KUKA KRL program: Station500_SprueCutter.src, Station500_SprueCutter.dat

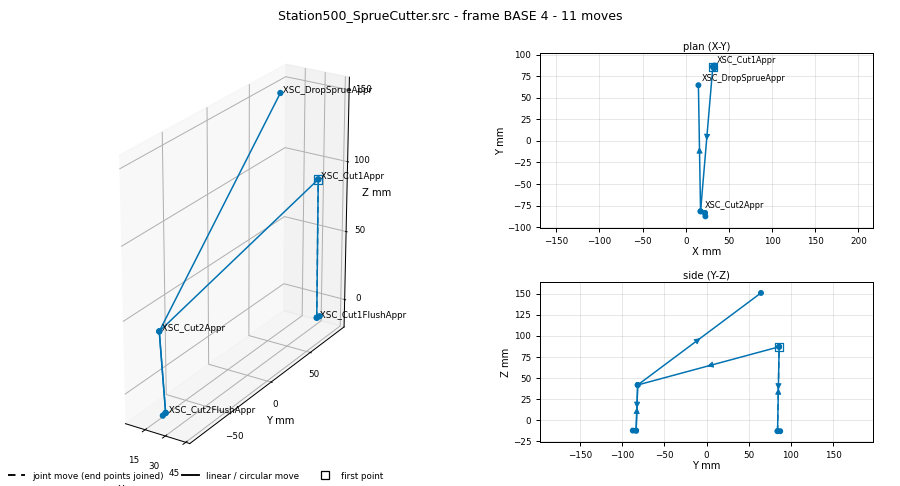
[picture p0: tool path of Station500_SprueCutter.src in frame BASE 4, 11 of 18 moves have a stored position in this frame; points joined in program order, loops and branches not executed]
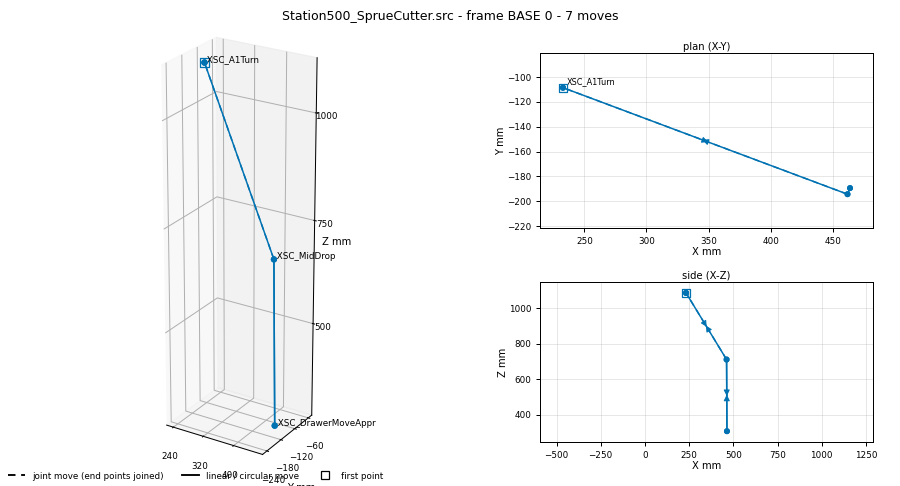
[picture p1: tool path of Station500_SprueCutter.src in frame BASE 0, 7 of 18 moves have a stored position in this frame; points joined in program order, loops and branches not executed]
--- Station500_SprueCutter.src ---
&ACCESS RVO1
&REL 8
&PARAM DISKPATH = KRC:\R1\Program
DEF Station500_SprueCutter()
   ;FOLD INI;%{PE}
      ;FOLD BASISTECH INI
         GLOBAL INTERRUPT DECL 3 WHEN $STOPMESS == TRUE DO IR_STOPM()
         INTERRUPT ON 3
         BAS(#INITMOV, 0)
      ;ENDFOLD (BASISTECH INI)
      ;FOLD USER INI
         ;Make your modifications here
      ;ENDFOLD (USER INI)
   ;ENDFOLD (INI)
;FOLD SPTP SC_A1Turn Vel=100 % PDAT2 Tool[0] Base[0] ;%{PE}
;FOLD Parameters ;%{h}
;Params IlfProvider=kukaroboter.basistech.inlineforms.movement.spline; Kuka.IsGlobalPoint=False; Kuka.PointName=SC_A1Turn; Kuka.BlendingEnabled=False; Kuka.MoveDataPtpName=PDAT2; Kuka.VelocityPtp=100; Kuka.VelocityFieldEnabled=True; Kuka.ColDetectFieldEnabled=True; Kuka.CurrentCDSetIndex=0; Kuka.MovementParameterFieldEnabled=True; IlfCommand=SPTP
;ENDFOLD
SPTP XSC_A1Turn WITH $VEL_AXIS[1] = SVEL_JOINT(100.0), $TOOL = STOOL2(FSC_A1Turn), $BASE = SBASE(FSC_A1Turn.BASE_NO), $IPO_MODE = SIPO_MODE(FSC_A1Turn.IPO_FRAME), $LOAD = SLOAD(FSC_A1Turn.TOOL_NO), $ACC_AXIS[1] = SACC_JOINT(PPDAT2), $APO = SAPO_PTP(PPDAT2), $GEAR_JERK[1] = SGEAR_JERK(PPDAT2), $COLLMON_TOL_PRO[1] = USE_CM_PRO_VALUES(0)
;ENDFOLD

   ;FOLD SPTP SC_Cut1Appr Vel=100 % PDAT4 Tool[2]:TOOL_DATA[2] Base[4]:BASE_DATA[4] ;%{PE}
      ;FOLD Parameters ;%{h}
         ;Params IlfProvider=kukaroboter.basistech.inlineforms.movement.spline; Kuka.IsGlobalPoint=False; Kuka.PointName=SC_Cut1Appr; Kuka.BlendingEnabled=False; Kuka.MoveDataPtpName=PDAT4; Kuka.VelocityPtp=100; Kuka.VelocityFieldEnabled=True; Kuka.ColDetectFieldEnabled=True; Kuka.CurrentCDSetIndex=0; Kuka.MovementParameterFieldEnabled=True; IlfCommand=SPTP; SimId=
      ;ENDFOLD
      SPTP XSC_Cut1Appr WITH $VEL_AXIS[1] = SVEL_JOINT(100.0), $TOOL = STOOL2(FSC_Cut1Appr), $BASE = SBASE(FSC_Cut1Appr.BASE_NO), $IPO_MODE = SIPO_MODE(FSC_Cut1Appr.IPO_FRAME), $LOAD = SLOAD(FSC_Cut1Appr.TOOL_NO), $ACC_AXIS[1] = SACC_JOINT(PPDAT4), $APO = SAPO_PTP(PPDAT4), $GEAR_JERK[1] = SGEAR_JERK(PPDAT4), $COLLMON_TOL_PRO[1] = USE_CM_PRO_VALUES(0)
      ;ENDFOLD

   ;FOLD SLIN SC_Cut1FlushAppr Vel=0.2 m/s CPDAT8 Tool[2]:TOOL_DATA[2] Base[4]:BASE_DATA[4] ;%{PE}
      ;FOLD Parameters ;%{h}
         ;Params IlfProvider=kukaroboter.basistech.inlineforms.movement.spline; Kuka.IsGlobalPoint=False; Kuka.PointName=SC_Cut1FlushAppr; Kuka.BlendingEnabled=False; Kuka.MoveDataName=CPDAT8; Kuka.VelocityPath=0.2; Kuka.VelocityFieldEnabled=True; Kuka.ColDetectFieldEnabled=True; Kuka.CurrentCDSetIndex=0; Kuka.MovementParameterFieldEnabled=True; IlfCommand=SLIN; SimId=
      ;ENDFOLD
      SLIN XSC_Cut1FlushAppr WITH $VEL = SVEL_CP(0.2, , LCPDAT8), $TOOL = STOOL2(FSC_Cut1FlushAppr), $BASE = SBASE(FSC_Cut1FlushAppr.BASE_NO), $IPO_MODE = SIPO_MODE(FSC_Cut1FlushAppr.IPO_FRAME), $LOAD = SLOAD(FSC_Cut1FlushAppr.TOOL_NO), $ACC = SACC_CP(LCPDAT8), $ORI_TYPE = SORI_TYP(LCPDAT8), $APO = SAPO(LCPDAT8), $JERK = SJERK(LCPDAT8), $COLLMON_TOL_PRO[1] = USE_CM_PRO_VALUES(0)
      ;ENDFOLD

   ;FOLD SLIN SC_Cut1Flush Vel=0.1 m/s CPDAT5 Tool[2]:TOOL_DATA[2] Base[4]:BASE_DATA[4] ;%{PE}
      ;FOLD Parameters ;%{h}
         ;Params IlfProvider=kukaroboter.basistech.inlineforms.movement.spline; Kuka.IsGlobalPoint=False; Kuka.PointName=SC_Cut1Flush; Kuka.BlendingEnabled=False; Kuka.MoveDataName=CPDAT5; Kuka.VelocityPath=0.1; Kuka.VelocityFieldEnabled=True; Kuka.ColDetectFieldEnabled=True; Kuka.CurrentCDSetIndex=0; Kuka.MovementParameterFieldEnabled=True; IlfCommand=SLIN; SimId=
      ;ENDFOLD
      SLIN XSC_Cut1Flush WITH $VEL = SVEL_CP(0.1, , LCPDAT5), $TOOL = STOOL2(FSC_Cut1Flush), $BASE = SBASE(FSC_Cut1Flush.BASE_NO), $IPO_MODE = SIPO_MODE(FSC_Cut1Flush.IPO_FRAME), $LOAD = SLOAD(FSC_Cut1Flush.TOOL_NO), $ACC = SACC_CP(LCPDAT5), $ORI_TYPE = SORI_TYP(LCPDAT5), $APO = SAPO(LCPDAT5), $JERK = SJERK(LCPDAT5), $COLLMON_TOL_PRO[1] = USE_CM_PRO_VALUES(0)
      ;ENDFOLD

RtoPLC_SprueCut1=True
    Wait Sec .25
RtoPLC_SprueCut1=False
    Wait Sec .25
   ;FOLD SLIN SC_Cut1FlushAppr Vel=0.2 m/s CPDAT8 Tool[2]:TOOL_DATA[2] Base[4]:BASE_DATA[4] ;%{PE}
      ;FOLD Parameters ;%{h}
         ;Params IlfProvider=kukaroboter.basistech.inlineforms.movement.spline; Kuka.IsGlobalPoint=False; Kuka.PointName=SC_Cut1FlushAppr; Kuka.BlendingEnabled=False; Kuka.MoveDataName=CPDAT8; Kuka.VelocityPath=0.2; Kuka.VelocityFieldEnabled=True; Kuka.ColDetectFieldEnabled=True; Kuka.CurrentCDSetIndex=0; Kuka.MovementParameterFieldEnabled=True; IlfCommand=SLIN; SimId=
      ;ENDFOLD
      SLIN XSC_Cut1FlushAppr WITH $VEL = SVEL_CP(0.2, , LCPDAT8), $TOOL = STOOL2(FSC_Cut1FlushAppr), $BASE = SBASE(FSC_Cut1FlushAppr.BASE_NO), $IPO_MODE = SIPO_MODE(FSC_Cut1FlushAppr.IPO_FRAME), $LOAD = SLOAD(FSC_Cut1FlushAppr.TOOL_NO), $ACC = SACC_CP(LCPDAT8), $ORI_TYPE = SORI_TYP(LCPDAT8), $APO = SAPO(LCPDAT8), $JERK = SJERK(LCPDAT8), $COLLMON_TOL_PRO[1] = USE_CM_PRO_VALUES(0)
      ;ENDFOLD

   ;FOLD SPTP SC_Cut1Appr Vel=100 % PDAT4 Tool[2]:TOOL_DATA[2] Base[4]:BASE_DATA[4] ;%{PE}
      ;FOLD Parameters ;%{h}
         ;Params IlfProvider=kukaroboter.basistech.inlineforms.movement.spline; Kuka.IsGlobalPoint=False; Kuka.PointName=SC_Cut1Appr; Kuka.BlendingEnabled=False; Kuka.MoveDataPtpName=PDAT4; Kuka.VelocityPtp=100; Kuka.VelocityFieldEnabled=True; Kuka.ColDetectFieldEnabled=True; Kuka.CurrentCDSetIndex=0; Kuka.MovementParameterFieldEnabled=True; IlfCommand=SPTP; SimId=
      ;ENDFOLD
      SPTP XSC_Cut1Appr WITH $VEL_AXIS[1] = SVEL_JOINT(100.0), $TOOL = STOOL2(FSC_Cut1Appr), $BASE = SBASE(FSC_Cut1Appr.BASE_NO), $IPO_MODE = SIPO_MODE(FSC_Cut1Appr.IPO_FRAME), $LOAD = SLOAD(FSC_Cut1Appr.TOOL_NO), $ACC_AXIS[1] = SACC_JOINT(PPDAT4), $APO = SAPO_PTP(PPDAT4), $GEAR_JERK[1] = SGEAR_JERK(PPDAT4), $COLLMON_TOL_PRO[1] = USE_CM_PRO_VALUES(0)
      ;ENDFOLD

   ;FOLD SLIN SC_Cut2Appr Vel=2 m/s CPDAT3 Tool[2]:TOOL_DATA[2] Base[4]:BASE_DATA[4] ;%{PE}
      ;FOLD Parameters ;%{h}
         ;Params IlfProvider=kukaroboter.basistech.inlineforms.movement.spline; Kuka.IsGlobalPoint=False; Kuka.PointName=SC_Cut2Appr; Kuka.BlendingEnabled=False; Kuka.MoveDataName=CPDAT3; Kuka.VelocityPath=2; Kuka.VelocityFieldEnabled=True; Kuka.ColDetectFieldEnabled=True; Kuka.CurrentCDSetIndex=0; Kuka.MovementParameterFieldEnabled=True; IlfCommand=SLIN; SimId=
      ;ENDFOLD
      SLIN XSC_Cut2Appr WITH $VEL = SVEL_CP(2.0, , LCPDAT3), $TOOL = STOOL2(FSC_Cut2Appr), $BASE = SBASE(FSC_Cut2Appr.BASE_NO), $IPO_MODE = SIPO_MODE(FSC_Cut2Appr.IPO_FRAME), $LOAD = SLOAD(FSC_Cut2Appr.TOOL_NO), $ACC = SACC_CP(LCPDAT3), $ORI_TYPE = SORI_TYP(LCPDAT3), $APO = SAPO(LCPDAT3), $JERK = SJERK(LCPDAT3), $COLLMON_TOL_PRO[1] = USE_CM_PRO_VALUES(0)
      ;ENDFOLD

   ;FOLD SLIN SC_Cut2FlushAppr Vel=0.2 m/s CPDAT10 Tool[2]:TOOL_DATA[2] Base[4]:BASE_DATA[4] ;%{PE}
      ;FOLD Parameters ;%{h}
         ;Params IlfProvider=kukaroboter.basistech.inlineforms.movement.spline; Kuka.IsGlobalPoint=False; Kuka.PointName=SC_Cut2FlushAppr; Kuka.BlendingEnabled=False; Kuka.MoveDataName=CPDAT10; Kuka.VelocityPath=0.2; Kuka.VelocityFieldEnabled=True; Kuka.ColDetectFieldEnabled=True; Kuka.CurrentCDSetIndex=0; Kuka.MovementParameterFieldEnabled=True; IlfCommand=SLIN; SimId=
      ;ENDFOLD
      SLIN XSC_Cut2FlushAppr WITH $VEL = SVEL_CP(0.2, , LCPDAT10), $TOOL = STOOL2(FSC_Cut2FlushAppr), $BASE = SBASE(FSC_Cut2FlushAppr.BASE_NO), $IPO_MODE = SIPO_MODE(FSC_Cut2FlushAppr.IPO_FRAME), $LOAD = SLOAD(FSC_Cut2FlushAppr.TOOL_NO), $ACC = SACC_CP(LCPDAT10), $ORI_TYPE = SORI_TYP(LCPDAT10), $APO = SAPO(LCPDAT10), $JERK = SJERK(LCPDAT10), $COLLMON_TOL_PRO[1] = USE_CM_PRO_VALUES(0)
      ;ENDFOLD

   ;FOLD SLIN SC_Cut2Flush Vel=0.1 m/s CPDAT2 Tool[2]:TOOL_DATA[2] Base[4]:BASE_DATA[4] ;%{PE}
      ;FOLD Parameters ;%{h}
         ;Params IlfProvider=kukaroboter.basistech.inlineforms.movement.spline; Kuka.IsGlobalPoint=False; Kuka.PointName=SC_Cut2Flush; Kuka.BlendingEnabled=False; Kuka.MoveDataName=CPDAT2; Kuka.VelocityPath=0.1; Kuka.VelocityFieldEnabled=True; Kuka.ColDetectFieldEnabled=True; Kuka.CurrentCDSetIndex=0; Kuka.MovementParameterFieldEnabled=True; IlfCommand=SLIN; SimId=
      ;ENDFOLD
      SLIN XSC_Cut2Flush WITH $VEL = SVEL_CP(0.1, , LCPDAT2), $TOOL = STOOL2(FSC_Cut2Flush), $BASE = SBASE(FSC_Cut2Flush.BASE_NO), $IPO_MODE = SIPO_MODE(FSC_Cut2Flush.IPO_FRAME), $LOAD = SLOAD(FSC_Cut2Flush.TOOL_NO), $ACC = SACC_CP(LCPDAT2), $ORI_TYPE = SORI_TYP(LCPDAT2), $APO = SAPO(LCPDAT2), $JERK = SJERK(LCPDAT2), $COLLMON_TOL_PRO[1] = USE_CM_PRO_VALUES(0)
      ;ENDFOLD
RtoPLC_SprueCut2=True
    Wait Sec .25
RtoPLC_SprueCut2=False
    Wait Sec .25
   ;FOLD SLIN SC_Cut2FlushAppr Vel=0.2 m/s CPDAT10 Tool[2]:TOOL_DATA[2] Base[4]:BASE_DATA[4] ;%{PE}
      ;FOLD Parameters ;%{h}
         ;Params IlfProvider=kukaroboter.basistech.inlineforms.movement.spline; Kuka.IsGlobalPoint=False; Kuka.PointName=SC_Cut2FlushAppr; Kuka.BlendingEnabled=False; Kuka.MoveDataName=CPDAT10; Kuka.VelocityPath=0.2; Kuka.VelocityFieldEnabled=True; Kuka.ColDetectFieldEnabled=True; Kuka.CurrentCDSetIndex=0; Kuka.MovementParameterFieldEnabled=True; IlfCommand=SLIN; SimId=
      ;ENDFOLD
      SLIN XSC_Cut2FlushAppr WITH $VEL = SVEL_CP(0.2, , LCPDAT10), $TOOL = STOOL2(FSC_Cut2FlushAppr), $BASE = SBASE(FSC_Cut2FlushAppr.BASE_NO), $IPO_MODE = SIPO_MODE(FSC_Cut2FlushAppr.IPO_FRAME), $LOAD = SLOAD(FSC_Cut2FlushAppr.TOOL_NO), $ACC = SACC_CP(LCPDAT10), $ORI_TYPE = SORI_TYP(LCPDAT10), $APO = SAPO(LCPDAT10), $JERK = SJERK(LCPDAT10), $COLLMON_TOL_PRO[1] = USE_CM_PRO_VALUES(0)
      ;ENDFOLD

         ;FOLD SLIN SC_Cut2Appr Vel=2 m/s CPDAT3 Tool[2]:TOOL_DATA[2] Base[4]:BASE_DATA[4] ;%{PE}
      ;FOLD Parameters ;%{h}
         ;Params IlfProvider=kukaroboter.basistech.inlineforms.movement.spline; Kuka.IsGlobalPoint=False; Kuka.PointName=SC_Cut2Appr; Kuka.BlendingEnabled=False; Kuka.MoveDataName=CPDAT3; Kuka.VelocityPath=2; Kuka.VelocityFieldEnabled=True; Kuka.ColDetectFieldEnabled=True; Kuka.CurrentCDSetIndex=0; Kuka.MovementParameterFieldEnabled=True; IlfCommand=SLIN; SimId=
      ;ENDFOLD
      SLIN XSC_Cut2Appr WITH $VEL = SVEL_CP(2.0, , LCPDAT3), $TOOL = STOOL2(FSC_Cut2Appr), $BASE = SBASE(FSC_Cut2Appr.BASE_NO), $IPO_MODE = SIPO_MODE(FSC_Cut2Appr.IPO_FRAME), $LOAD = SLOAD(FSC_Cut2Appr.TOOL_NO), $ACC = SACC_CP(LCPDAT3), $ORI_TYPE = SORI_TYP(LCPDAT3), $APO = SAPO(LCPDAT3), $JERK = SJERK(LCPDAT3), $COLLMON_TOL_PRO[1] = USE_CM_PRO_VALUES(0)
      ;ENDFOLD

   ;FOLD SLIN SC_DropSprueAppr Vel=2 m/s CPDAT14 Tool[2]:TOOL_DATA[2] Base[4]:BASE_DATA[4] ;%{PE}
      ;FOLD Parameters ;%{h}
         ;Params IlfProvider=kukaroboter.basistech.inlineforms.movement.spline; Kuka.IsGlobalPoint=False; Kuka.PointName=SC_DropSprueAppr; Kuka.BlendingEnabled=False; Kuka.MoveDataName=CPDAT14; Kuka.VelocityPath=2; Kuka.VelocityFieldEnabled=True; Kuka.ColDetectFieldEnabled=True; Kuka.CurrentCDSetIndex=0; Kuka.MovementParameterFieldEnabled=True; IlfCommand=SLIN
      ;ENDFOLD
      SLIN XSC_DropSprueAppr WITH $VEL = SVEL_CP(2.0, , LCPDAT14), $TOOL = STOOL2(FSC_DropSprueAppr), $BASE = SBASE(FSC_DropSprueAppr.BASE_NO), $IPO_MODE = SIPO_MODE(FSC_DropSprueAppr.IPO_FRAME), $LOAD = SLOAD(FSC_DropSprueAppr.TOOL_NO), $ACC = SACC_CP(LCPDAT14), $ORI_TYPE = SORI_TYP(LCPDAT14), $APO = SAPO(LCPDAT14), $JERK = SJERK(LCPDAT14), $COLLMON_TOL_PRO[1] = USE_CM_PRO_VALUES(0)
      ;ENDFOLD
RtoPLC_FinishGripClose=False
wait sec .5
RtoPLC_FinishGripOpen=True
    Wait Sec .25
RtoPLC_FinishGripOpen=False
    Wait Sec .25

   ;FOLD SPTP SC_A1Return Vel=100 % PDAT3 Tool[0] Base[0] ;%{PE}
      ;FOLD Parameters ;%{h}
         ;Params IlfProvider=kukaroboter.basistech.inlineforms.movement.spline; Kuka.IsGlobalPoint=False; Kuka.PointName=SC_A1Return; Kuka.BlendingEnabled=False; Kuka.MoveDataPtpName=PDAT3; Kuka.VelocityPtp=100; Kuka.VelocityFieldEnabled=True; Kuka.ColDetectFieldEnabled=True; Kuka.CurrentCDSetIndex=0; Kuka.MovementParameterFieldEnabled=True; IlfCommand=SPTP
      ;ENDFOLD
      SPTP XSC_A1Return WITH $VEL_AXIS[1] = SVEL_JOINT(100.0), $TOOL = STOOL2(FSC_A1Return), $BASE = SBASE(FSC_A1Return.BASE_NO), $IPO_MODE = SIPO_MODE(FSC_A1Return.IPO_FRAME), $LOAD = SLOAD(FSC_A1Return.TOOL_NO), $ACC_AXIS[1] = SACC_JOINT(PPDAT3), $APO = SAPO_PTP(PPDAT3), $GEAR_JERK[1] = SGEAR_JERK(PPDAT3), $COLLMON_TOL_PRO[1] = USE_CM_PRO_VALUES(0)
      ;ENDFOLD

;Check for drawer full
If PLCtoR_DrawerFull==True Then

;FOLD SLIN SC_MidDrop Vel=2 m/s CPDAT17 Tool[0] Base[0] ;%{PE}
;FOLD Parameters ;%{h}
;Params IlfProvider=kukaroboter.basistech.inlineforms.movement.spline; Kuka.IsGlobalPoint=False; Kuka.PointName=SC_MidDrop; Kuka.BlendingEnabled=False; Kuka.MoveDataName=CPDAT17; Kuka.VelocityPath=2; Kuka.VelocityFieldEnabled=True; Kuka.ColDetectFieldEnabled=True; Kuka.CurrentCDSetIndex=0; Kuka.MovementParameterFieldEnabled=True; IlfCommand=SLIN
;ENDFOLD
SLIN XSC_MidDrop WITH $VEL = SVEL_CP(2.0, , LCPDAT17), $TOOL = STOOL2(FSC_MidDrop), $BASE = SBASE(FSC_MidDrop.BASE_NO), $IPO_MODE = SIPO_MODE(FSC_MidDrop.IPO_FRAME), $LOAD = SLOAD(FSC_MidDrop.TOOL_NO), $ACC = SACC_CP(LCPDAT17), $ORI_TYPE = SORI_TYP(LCPDAT17), $APO = SAPO(LCPDAT17), $JERK = SJERK(LCPDAT17), $COLLMON_TOL_PRO[1] = USE_CM_PRO_VALUES(0)
;ENDFOLD

;FOLD SLIN SC_DrawerMoveAppr Vel=2 m/s CPDAT18 Tool[0] Base[0] ;%{PE}
;FOLD Parameters ;%{h}
;Params IlfProvider=kukaroboter.basistech.inlineforms.movement.spline; Kuka.IsGlobalPoint=False; Kuka.PointName=SC_DrawerMoveAppr; Kuka.BlendingEnabled=False; Kuka.MoveDataName=CPDAT18; Kuka.VelocityPath=2; Kuka.VelocityFieldEnabled=True; Kuka.ColDetectFieldEnabled=True; Kuka.CurrentCDSetIndex=0; Kuka.MovementParameterFieldEnabled=True; IlfCommand=SLIN
;ENDFOLD
SLIN XSC_DrawerMoveAppr WITH $VEL = SVEL_CP(2.0, , LCPDAT18), $TOOL = STOOL2(FSC_DrawerMoveAppr), $BASE = SBASE(FSC_DrawerMoveAppr.BASE_NO), $IPO_MODE = SIPO_MODE(FSC_DrawerMoveAppr.IPO_FRAME), $LOAD = SLOAD(FSC_DrawerMoveAppr.TOOL_NO), $ACC = SACC_CP(LCPDAT18), $ORI_TYPE = SORI_TYP(LCPDAT18), $APO = SAPO(LCPDAT18), $JERK = SJERK(LCPDAT18), $COLLMON_TOL_PRO[1] = USE_CM_PRO_VALUES(0)
;ENDFOLD

Station500_DrawerMove()

;FOLD SLIN SC_DrawerMoveAppr Vel=2 m/s CPDAT18 Tool[0] Base[0] ;%{PE}
;FOLD Parameters ;%{h}
;Params IlfProvider=kukaroboter.basistech.inlineforms.movement.spline; Kuka.IsGlobalPoint=False; Kuka.PointName=SC_DrawerMoveAppr; Kuka.BlendingEnabled=False; Kuka.MoveDataName=CPDAT18; Kuka.VelocityPath=2; Kuka.VelocityFieldEnabled=True; Kuka.ColDetectFieldEnabled=True; Kuka.CurrentCDSetIndex=0; Kuka.MovementParameterFieldEnabled=True; IlfCommand=SLIN
;ENDFOLD
SLIN XSC_DrawerMoveAppr WITH $VEL = SVEL_CP(2.0, , LCPDAT18), $TOOL = STOOL2(FSC_DrawerMoveAppr), $BASE = SBASE(FSC_DrawerMoveAppr.BASE_NO), $IPO_MODE = SIPO_MODE(FSC_DrawerMoveAppr.IPO_FRAME), $LOAD = SLOAD(FSC_DrawerMoveAppr.TOOL_NO), $ACC = SACC_CP(LCPDAT18), $ORI_TYPE = SORI_TYP(LCPDAT18), $APO = SAPO(LCPDAT18), $JERK = SJERK(LCPDAT18), $COLLMON_TOL_PRO[1] = USE_CM_PRO_VALUES(0)
;ENDFOLD

;FOLD SLIN SC_MidDrop Vel=2 m/s CPDAT17 Tool[0] Base[0] ;%{PE}
;FOLD Parameters ;%{h}
;Params IlfProvider=kukaroboter.basistech.inlineforms.movement.spline; Kuka.IsGlobalPoint=False; Kuka.PointName=SC_MidDrop; Kuka.BlendingEnabled=False; Kuka.MoveDataName=CPDAT17; Kuka.VelocityPath=2; Kuka.VelocityFieldEnabled=True; Kuka.ColDetectFieldEnabled=True; Kuka.CurrentCDSetIndex=0; Kuka.MovementParameterFieldEnabled=True; IlfCommand=SLIN
;ENDFOLD
SLIN XSC_MidDrop WITH $VEL = SVEL_CP(2.0, , LCPDAT17), $TOOL = STOOL2(FSC_MidDrop), $BASE = SBASE(FSC_MidDrop.BASE_NO), $IPO_MODE = SIPO_MODE(FSC_MidDrop.IPO_FRAME), $LOAD = SLOAD(FSC_MidDrop.TOOL_NO), $ACC = SACC_CP(LCPDAT17), $ORI_TYPE = SORI_TYP(LCPDAT17), $APO = SAPO(LCPDAT17), $JERK = SJERK(LCPDAT17), $COLLMON_TOL_PRO[1] = USE_CM_PRO_VALUES(0)
;ENDFOLD



RtoPLC_DrawerIsFullWarn=True
wait sec .5
RtoPLC_DrawerIsFullWarn=False
EndIf



;FOLD SPTP SC_A1Return Vel=100 % PDAT15 Tool[0] Base[0] ;%{PE}
;FOLD Parameters ;%{h}
;Params IlfProvider=kukaroboter.basistech.inlineforms.movement.spline; Kuka.IsGlobalPoint=False; Kuka.PointName=SC_A1Return; Kuka.BlendingEnabled=False; Kuka.MoveDataPtpName=PDAT15; Kuka.VelocityPtp=100; Kuka.VelocityFieldEnabled=True; Kuka.ColDetectFieldEnabled=True; Kuka.CurrentCDSetIndex=0; Kuka.MovementParameterFieldEnabled=True; IlfCommand=SPTP
;ENDFOLD
SPTP XSC_A1Return WITH $VEL_AXIS[1] = SVEL_JOINT(100.0), $TOOL = STOOL2(FSC_A1Return), $BASE = SBASE(FSC_A1Return.BASE_NO), $IPO_MODE = SIPO_MODE(FSC_A1Return.IPO_FRAME), $LOAD = SLOAD(FSC_A1Return.TOOL_NO), $ACC_AXIS[1] = SACC_JOINT(PPDAT15), $APO = SAPO_PTP(PPDAT15), $GEAR_JERK[1] = SGEAR_JERK(PPDAT15), $COLLMON_TOL_PRO[1] = USE_CM_PRO_VALUES(0)
;ENDFOLD
Wait For PLCtoR_DrawerInPos==True

END

--- Station500_SprueCutter.dat ---
&ACCESS  RVP
&PARAM DISKPATH = KRC:\R1\Program
&REL 8
DEFDAT  STATION500_SPRUECUTTER
;FOLD EXTERNAL DECLARATIONS;%{PE}%MKUKATPBASIS,%CEXT,%VCOMMON,%P
;FOLD BASISTECH EXT;%{PE}%MKUKATPBASIS,%CEXT,%VEXT,%P
EXT  BAS (BAS_COMMAND  :IN,REAL  :IN )
DECL INT SUCCESS
;ENDFOLD (BASISTECH EXT)
;FOLD USER EXT;%{E}%MKUKATPUSER,%CEXT,%VEXT,%P
;Make your modifications here

;ENDFOLD (USER EXT)
;ENDFOLD (EXTERNAL DECLARATIONS)
DECL PDAT PPDAT1={VEL 100.000,ACC 60.0000,APO_DIST 500.000,APO_MODE #CDIS,GEAR_JERK 100.000,EXAX_IGN 0}
DECL LDAT LCPDAT1={VEL 2.00000,ACC 60.0000,APO_DIST 500.000,APO_FAC 50.0000,AXIS_VEL 100.000,AXIS_ACC 60.0000,ORI_TYP #VAR,CIRC_TYP #BASE,JERK_FAC 50.0000,GEAR_JERK 100.000,EXAX_IGN 0}
DECL E6POS XSC_Cut1Appr={X 31.4316330,Y 85.9856110,Z 87.1636124,A -8.00368690,B -1.05840850,C 179.069397,S 2,T 10,E1 0.0,E2 0.0,E3 0.0,E4 0.0,E5 0.0,E6 0.0}
DECL FDAT FSC_Cut1Appr={TOOL_NO 2,BASE_NO 4,IPO_FRAME #BASE,POINT2[] " "}
DECL LDAT LCPDAT2={VEL 0.100000,ACC 60.0000,APO_DIST 500.000,APO_FAC 50.0000,AXIS_VEL 100.000,AXIS_ACC 60.0000,ORI_TYP #VAR,CIRC_TYP #BASE,JERK_FAC 50.0000,GEAR_JERK 100.000,EXAX_IGN 0}
DECL LDAT LCPDAT3={VEL 2.00000,ACC 60.0000,APO_DIST 500.000,APO_FAC 50.0000,AXIS_VEL 100.000,AXIS_ACC 60.0000,ORI_TYP #VAR,CIRC_TYP #BASE,JERK_FAC 50.0000,GEAR_JERK 100.000,EXAX_IGN 0}
DECL E6POS XSC_Cut2Appr={X 17.2129917,Y -81.6377182,Z 41.9165344,A 8.14923,B -0.756849885,C 178.816269,S 2,T 2,E1 0.0,E2 0.0,E3 0.0,E4 0.0,E5 0.0,E6 0.0}
DECL FDAT FSC_Cut2Appr={TOOL_NO 2,BASE_NO 4,IPO_FRAME #BASE,POINT2[] " "}
DECL PDAT PDEFAULT={VEL 100.000,ACC 60.0000,APO_DIST 500.000,APO_MODE #CDIS,GEAR_JERK 100.000,EXAX_IGN 0}
DECL PDAT PPDAT2={VEL 100.000,ACC 100.000,APO_DIST 500.000,APO_MODE #CDIS,GEAR_JERK 100.000,EXAX_IGN 0}
DECL PDAT PPDAT3={VEL 100.000,ACC 60.0000,APO_DIST 500.000,APO_MODE #CDIS,GEAR_JERK 100.000,EXAX_IGN 0}
DECL LDAT LCPDAT4={VEL 2.00000,ACC 60.0000,APO_DIST 500.000,APO_FAC 50.0000,AXIS_VEL 100.000,AXIS_ACC 60.0000,ORI_TYP #VAR,CIRC_TYP #BASE,JERK_FAC 50.0000,GEAR_JERK 100.000,EXAX_IGN 0}
DECL PDAT PPDAT4={VEL 100.000,ACC 60.0000,APO_DIST 500.000,APO_MODE #CDIS,GEAR_JERK 100.000,EXAX_IGN 0}
DECL PDAT PPDAT5={VEL 100.000,ACC 60.0000,APO_DIST 500.000,APO_MODE #CDIS,GEAR_JERK 100.000,EXAX_IGN 0}
DECL LDAT LCPDAT5={VEL 0.100000,ACC 60.0000,APO_DIST 500.000,APO_FAC 50.0000,AXIS_VEL 100.000,AXIS_ACC 60.0000,ORI_TYP #VAR,CIRC_TYP #BASE,JERK_FAC 50.0000,GEAR_JERK 100.000,EXAX_IGN 0}
DECL LDAT LCPDAT6={VEL 0.200000,ACC 60.0000,APO_DIST 500.000,APO_FAC 50.0000,AXIS_VEL 100.000,AXIS_ACC 60.0000,ORI_TYP #VAR,CIRC_TYP #BASE,JERK_FAC 50.0000,GEAR_JERK 100.000,EXAX_IGN 0}
DECL E6POS XSC_Cut1Return={X 19.8408470,Y 89.1498413,Z 88.3440094,A -2.79877567,B -0.969627,C 178.977219,S 2,T 10,E1 0.0,E2 0.0,E3 0.0,E4 0.0,E5 0.0,E6 0.0}
DECL FDAT FSC_Cut1Return={TOOL_NO 2,BASE_NO 4,IPO_FRAME #BASE,POINT2[] " "}
DECL LDAT LCPDAT7={VEL 0.200000,ACC 60.0000,APO_DIST 500.000,APO_FAC 50.0000,AXIS_VEL 100.000,AXIS_ACC 60.0000,ORI_TYP #VAR,CIRC_TYP #BASE,JERK_FAC 50.0000,GEAR_JERK 100.000,EXAX_IGN 0}
DECL E6POS XSC_Cut2Return={X 16.9239788,Y -85.9609451,Z -9.08849,A 6.37688160,B -0.792611718,C 178.835648,S 2,T 2,E1 0.0,E2 0.0,E3 0.0,E4 0.0,E5 0.0,E6 0.0}
DECL FDAT FSC_Cut2Return={TOOL_NO 2,BASE_NO 4,IPO_FRAME #BASE,POINT2[] " "}
DECL LDAT LCPDAT8={VEL 0.200000,ACC 60.0000,APO_DIST 500.000,APO_FAC 50.0000,AXIS_VEL 100.000,AXIS_ACC 60.0000,ORI_TYP #VAR,CIRC_TYP #BASE,JERK_FAC 50.0000,GEAR_JERK 100.000,EXAX_IGN 0}
DECL E6POS XSC_Cut1FlushAppr={X 33.0344238,Y 84.1201324,Z -12.8061390,A -8.00368690,B -1.05840850,C 179.069397,S 2,T 10,E1 0.0,E2 0.0,E3 0.0,E4 0.0,E5 0.0,E6 0.0}
DECL FDAT FSC_Cut1FlushAppr={TOOL_NO 2,BASE_NO 4,IPO_FRAME #BASE,POINT2[] " "}
DECL E6POS XSC_Cut1Flush={X 33.4769402,Y 87.2604752,Z -12.8576441,A -8.00368690,B -1.05840850,C 179.069397,S 2,T 10,E1 0.0,E2 0.0,E3 0.0,E4 0.0,E5 0.0,E6 0.0}
DECL FDAT FSC_Cut1Flush={TOOL_NO 2,BASE_NO 4,IPO_FRAME #BASE,POINT2[] " "}
DECL LDAT LCPDAT9={VEL 0.100000,ACC 60.0000,APO_DIST 500.000,APO_FAC 50.0000,AXIS_VEL 100.000,AXIS_ACC 60.0000,ORI_TYP #VAR,CIRC_TYP #BASE,JERK_FAC 50.0000,GEAR_JERK 100.000,EXAX_IGN 0}
DECL E6POS XSC_Cut1FlushReturn={X 21.4436378,Y 87.2843552,Z -11.6257420,A -2.79877567,B -0.969627,C 178.977219,S 2,T 10,E1 0.0,E2 0.0,E3 0.0,E4 0.0,E5 0.0,E6 0.0}
DECL FDAT FSC_Cut1FlushReturn={TOOL_NO 2,BASE_NO 4,IPO_FRAME #BASE,POINT2[] " "}
DECL LDAT LCPDAT10={VEL 0.200000,ACC 60.0000,APO_DIST 500.000,APO_FAC 50.0000,AXIS_VEL 100.000,AXIS_ACC 60.0000,ORI_TYP #VAR,CIRC_TYP #BASE,JERK_FAC 50.0000,GEAR_JERK 100.000,EXAX_IGN 0}
DECL E6POS XSC_Cut2FlushAppr={X 22.2581711,Y -83.4844055,Z -12.2257624,A 8.14923,B -0.756850123,C 178.816269,S 2,T 2,E1 0.0,E2 0.0,E3 0.0,E4 0.0,E5 0.0,E6 0.0}
DECL FDAT FSC_Cut2FlushAppr={TOOL_NO 2,BASE_NO 4,IPO_FRAME #BASE,POINT2[] " "}
DECL E6POS XSC_Cut2Flush={X 22.8239765,Y -87.4433212,Z -12.1431360,A 8.14923,B -0.756850064,C 178.816269,S 2,T 2,E1 0.0,E2 0.0,E3 0.0,E4 0.0,E5 0.0,E6 0.0}
DECL FDAT FSC_Cut2Flush={TOOL_NO 2,BASE_NO 4,IPO_FRAME #BASE,POINT2[] " "}
DECL LDAT LCPDAT11={VEL 0.100000,ACC 60.0000,APO_DIST 500.000,APO_FAC 50.0000,AXIS_VEL 100.000,AXIS_ACC 60.0000,ORI_TYP #VAR,CIRC_TYP #BASE,JERK_FAC 50.0000,GEAR_JERK 100.000,EXAX_IGN 0}
DECL E6POS XSC_Cut2FlushReturn={X 16.8861523,Y -86.2804108,Z -9.89605808,A 6.42420053,B -0.793163419,C 178.835037,S 2,T 2,E1 0.0,E2 0.0,E3 0.0,E4 0.0,E5 0.0,E6 0.0}
DECL FDAT FSC_Cut2FlushReturn={TOOL_NO 2,BASE_NO 4,IPO_FRAME #BASE,POINT2[] " "}
DECL PDAT PPDAT6={VEL 100.000,ACC 60.0000,APO_DIST 500.000,APO_MODE #CDIS,GEAR_JERK 100.000,EXAX_IGN 0}
DECL E6POS XSC_RejectFinishAppr={X 27.7327499,Y -365.697815,Z 105.706985,A 0.0136010,B -0.713825,C 178.914124,S 2,T 10,E1 0.0,E2 0.0,E3 0.0,E4 0.0,E5 0.0,E6 0.0}
DECL FDAT FSC_RejectFinishAppr={TOOL_NO 2,BASE_NO 4,IPO_FRAME #BASE,POINT2[] " "}
DECL PDAT PPDAT7={VEL 100.000,ACC 60.0000,APO_DIST 500.000,APO_MODE #CDIS,GEAR_JERK 100.000,EXAX_IGN 0}
DECL E6POS XSC_RejectFinishTilt={X 27.7327785,Y -365.697876,Z 105.706879,A 0.0136160,B -0.713835,C 148.914124,S 2,T 10,E1 0.0,E2 0.0,E3 0.0,E4 0.0,E5 0.0,E6 0.0}
DECL FDAT FSC_RejectFinishTilt={TOOL_NO 2,BASE_NO 4,IPO_FRAME #BASE,POINT2[] " "}
DECL PDAT PPDAT8={VEL 100.000,ACC 60.0000,APO_DIST 500.000,APO_MODE #CDIS,GEAR_JERK 100.000,EXAX_IGN 0}
DECL E6POS XSC_RejectFinishReturn={X 27.7327499,Y -365.697815,Z 105.706985,A 0.0136010,B -0.713825,C 178.914124,S 2,T 10,E1 0.0,E2 0.0,E3 0.0,E4 0.0,E5 0.0,E6 0.0}
DECL FDAT FSC_RejectFinishReturn={TOOL_NO 2,BASE_NO 4,IPO_FRAME #BASE,POINT2[] " "}
DECL PDAT PPDAT9={VEL 100.000,ACC 60.0000,APO_DIST 500.000,APO_MODE #CDIS,GEAR_JERK 100.000,EXAX_IGN 0}
DECL PDAT PPDAT10={VEL 100.000,ACC 60.0000,APO_DIST 500.000,APO_MODE #CDIS,GEAR_JERK 100.000,EXAX_IGN 0}
DECL E6POS XSC_A1Turn={X 232.779465,Y -108.546844,Z 1087.90991,A 154.999969,B 35.0000,C 179.999985,S 2,T 34,E1 0.0,E2 0.0,E3 0.0,E4 0.0,E5 0.0,E6 0.0}
DECL FDAT FSC_A1Turn={TOOL_NO 0,BASE_NO 0,IPO_FRAME #BASE,POINT2[] " "}
DECL E6POS XSC_A1Return={X 232.779465,Y -108.546844,Z 1087.90991,A 154.999969,B 35.0000,C 179.999985,S 2,T 34,E1 0.0,E2 0.0,E3 0.0,E4 0.0,E5 0.0,E6 0.0}
DECL FDAT FSC_A1Return={TOOL_NO 0,BASE_NO 0,IPO_FRAME #BASE,POINT2[] " "}
DECL E6POS XSC_RejectBlankAppr={X -38.9269943,Y -462.206268,Z 317.426,A 0.0137280,B -0.713833,C -1.08587503,S 2,T 10,E1 0.0,E2 0.0,E3 0.0,E4 0.0,E5 0.0,E6 0.0}
DECL FDAT FSC_RejectBlankAppr={TOOL_NO 1,BASE_NO 4,IPO_FRAME #BASE,POINT2[] " "}
DECL E6POS XSC_RejectBlankTilt={X -36.8766327,Y -465.324097,Z 152.922058,A 0.0137280,B -0.713833,C 23.9141254,S 2,T 34,E1 0.0,E2 0.0,E3 0.0,E4 0.0,E5 0.0,E6 0.0}
DECL FDAT FSC_RejectBlankTilt={TOOL_NO 1,BASE_NO 4,IPO_FRAME #BASE,POINT2[] " "}
DECL PDAT PPDAT11={VEL 100.000,ACC 60.0000,APO_DIST 500.000,APO_MODE #CDIS,GEAR_JERK 100.000,EXAX_IGN 0}
DECL PDAT PPDAT12={VEL 100.000,ACC 60.0000,APO_DIST 500.000,APO_MODE #CDIS,GEAR_JERK 100.000,EXAX_IGN 0}
DECL E6POS XSC_RejectBlankReturn={X -38.9269943,Y -462.206268,Z 317.426,A 0.0137280,B -0.713833,C -1.08587503,S 2,T 10,E1 0.0,E2 0.0,E3 0.0,E4 0.0,E5 0.0,E6 0.0}
DECL FDAT FSC_RejectBlankReturn={TOOL_NO 1,BASE_NO 4,IPO_FRAME #BASE,POINT2[] " "}
DECL E6POS XP1={X 232.779465,Y -108.546844,Z 1087.90991,A 154.999969,B 35.0000,C 179.999985,S 2,T 34,E1 0.0,E2 0.0,E3 0.0,E4 0.0,E5 0.0,E6 0.0}
DECL FDAT FP1={TOOL_NO 0,BASE_NO 0,IPO_FRAME #BASE,POINT2[] " "}
DECL PDAT PPDAT13={VEL 100.000,ACC 60.0000,APO_DIST 500.000,APO_MODE #CDIS,GEAR_JERK 100.000,EXAX_IGN 0}
DECL LDAT LCPDAT12={VEL 2.00000,ACC 60.0000,APO_DIST 500.000,APO_FAC 50.0000,AXIS_VEL 100.000,AXIS_ACC 60.0000,ORI_TYP #VAR,CIRC_TYP #BASE,JERK_FAC 50.0000,GEAR_JERK 100.000,EXAX_IGN 0}
DECL LDAT LCPDAT13={VEL 2.00000,ACC 60.0000,APO_DIST 500.000,APO_FAC 50.0000,AXIS_VEL 100.000,AXIS_ACC 60.0000,ORI_TYP #VAR,CIRC_TYP #BASE,JERK_FAC 50.0000,GEAR_JERK 100.000,EXAX_IGN 0}
DECL LDAT LCPDAT14={VEL 2.00000,ACC 60.0000,APO_DIST 500.000,APO_FAC 50.0000,AXIS_VEL 100.000,AXIS_ACC 60.0000,ORI_TYP #VAR,CIRC_TYP #BASE,JERK_FAC 50.0000,GEAR_JERK 100.000,EXAX_IGN 0}
DECL E6POS XSC_DropSprueAppr={X 14.7132511,Y 64.4652176,Z 150.976196,A 0.685273,B -32.2530365,C 88.7160645,S 2,T 10,E1 0.0,E2 0.0,E3 0.0,E4 0.0,E5 0.0,E6 0.0}
DECL FDAT FSC_DropSprueAppr={TOOL_NO 2,BASE_NO 4,IPO_FRAME #BASE,POINT2[] " "}
DECL FDAT FSC_Cut2FlushAppr_1={TOOL_NO 2,BASE_NO 4,IPO_FRAME #BASE,POINT2[] " "}
DECL LDAT LCPDAT15={VEL 0.200000,ACC 60.0000,APO_DIST 500.000,APO_FAC 50.0000,AXIS_VEL 100.000,AXIS_ACC 60.0000,ORI_TYP #VAR,CIRC_TYP #BASE,JERK_FAC 50.0000,GEAR_JERK 100.000,EXAX_IGN 0}
DECL E6POS XSC_Cut2FlushAppr_1={X 16.9239788,Y -85.9609451,Z -9.08849,A 6.37688160,B -0.792611718,C 178.835648,S 2,T 2,E1 0.0,E2 0.0,E3 0.0,E4 0.0,E5 0.0,E6 0.0}
DECL FDAT FSC_Cut2Appr_1={TOOL_NO 2,BASE_NO 4,IPO_FRAME #BASE,POINT2[] " "}
DECL LDAT LCPDAT16={VEL 2.00000,ACC 60.0000,APO_DIST 500.000,APO_FAC 50.0000,AXIS_VEL 100.000,AXIS_ACC 60.0000,ORI_TYP #VAR,CIRC_TYP #BASE,JERK_FAC 50.0000,GEAR_JERK 100.000,EXAX_IGN 0}
DECL E6POS XSC_Cut2Appr_1={X 15.3238029,Y -84.0951,Z 90.8812943,A 6.37688160,B -0.792611718,C 178.835648,S 2,T 10,E1 0.0,E2 0.0,E3 0.0,E4 0.0,E5 0.0,E6 0.0}
DECL MODULEPARAM_T LAST_TP_PARAMS={PARAMS[] "Kuka.VelocityFieldEnabled=True; Kuka.ColDetectFieldEnabled=True; Kuka.MovementParameterFieldEnabled=True; Kuka.IsAngleEnabled=False; Kuka.PointName=SC_A1Return; Kuka.FrameData.base_no=0; Kuka.FrameData.tool_no=0; Kuka.FrameData.ipo_frame=#BASE; Kuka.FrameData.point2=; Kuka.isglobalpoint=False; Kuka.MoveDataPtpName=PDAT15; Kuka.MovementDataPdat.apo_mode=#CDIS; Kuka.MovementDataPdat.apo_dist=500; Kuka.MovementData.vel=100; Kuka.MovementData.acc=35; Kuka.MovementData.exax_ign=0; Kuka.VelocityPtp=100; Kuka.BlendingEnabled=False; Kuka.APXEnabled=False; Kuka.CurrentCDSetIndex=0; Kuka.MoveDataName=CPDAT18; Kuka.MovementData.cb={AUX_PT {ORI #CONSIDER,E1 #CONSIDER,E2 #CONSIDER,E3 #CONSIDER,E4 #CONSIDER,E5 #CONSIDER,E6 #CONSIDER},TARGET_PT {ORI #INTERPOLATE,E1 #INTERPOLATE,E2 #INTERPOLATE,E3 #INTERPOLATE,E4 #INTERPOLATE,E5 #INTERPOLATE,E6 #INTERPOLATE}}; Kuka.MovementData.apo_fac=50; Kuka.MovementData.apo_dist=500; Kuka.MovementData.axis_acc=100; Kuka.MovementData.axis_vel=100; Kuka.MovementData.circ_typ=#BASE; Kuka.MovementData.jerk_fac=50; Kuka.MovementData.ori_typ=#VAR; Kuka.VelocityPath=2    "}
DECL E6POS XSC_MidDrop={X 461.954102,Y -194.353302,Z 711.295105,A 156.814987,B -0.00957452413,C 179.246414,S 2,T 42,E1 0.0,E2 0.0,E3 0.0,E4 0.0,E5 0.0,E6 0.0}
DECL FDAT FSC_MidDrop={TOOL_NO 0,BASE_NO 0,IPO_FRAME #BASE,POINT2[] " "}
DECL LDAT LCPDAT17={VEL 2.00000,ACC 100.000,APO_DIST 500.000,APO_FAC 50.0000,AXIS_VEL 100.000,AXIS_ACC 100.000,ORI_TYP #VAR,CIRC_TYP #BASE,JERK_FAC 50.0000,GEAR_JERK 100.000,EXAX_IGN 0,CB {AUX_PT {ORI #CONSIDER,E1 #CONSIDER,E2 #CONSIDER,E3 #CONSIDER,E4 #CONSIDER,E5 #CONSIDER,E6 #CONSIDER},TARGET_PT {ORI #INTERPOLATE,E1 #INTERPOLATE,E2 #INTERPOLATE,E3 #INTERPOLATE,E4 #INTERPOLATE,E5 #INTERPOLATE,E6 #INTERPOLATE}}}
DECL E6POS XSC_DrawerMoveAppr={X 463.991455,Y -189.424393,Z 305.849274,A 156.814987,B -0.00956464652,C 179.246399,S 2,T 10,E1 0.0,E2 0.0,E3 0.0,E4 0.0,E5 0.0,E6 0.0}
DECL FDAT FSC_DrawerMoveAppr={TOOL_NO 0,BASE_NO 0,IPO_FRAME #BASE,POINT2[] " "}
DECL LDAT LCPDAT18={VEL 2.00000,ACC 100.000,APO_DIST 500.000,APO_FAC 50.0000,AXIS_VEL 100.000,AXIS_ACC 100.000,ORI_TYP #VAR,CIRC_TYP #BASE,JERK_FAC 50.0000,GEAR_JERK 100.000,EXAX_IGN 0,CB {AUX_PT {ORI #CONSIDER,E1 #CONSIDER,E2 #CONSIDER,E3 #CONSIDER,E4 #CONSIDER,E5 #CONSIDER,E6 #CONSIDER},TARGET_PT {ORI #INTERPOLATE,E1 #INTERPOLATE,E2 #INTERPOLATE,E3 #INTERPOLATE,E4 #INTERPOLATE,E5 #INTERPOLATE,E6 #INTERPOLATE}}}
DECL PDAT PPDAT14={VEL 100.000,ACC 60.0000,APO_DIST 500.000,APO_MODE #CDIS,GEAR_JERK 100.000,EXAX_IGN 0}
DECL FDAT FSC_A1Return_1={TOOL_NO 0,BASE_NO 0,IPO_FRAME #BASE,POINT2[] " "}
DECL E6POS XSC_A1Return_1={X 232.779465,Y -108.546844,Z 1087.90991,A 154.999969,B 35.0000,C 179.999985,S 2,T 34,E1 0.0,E2 0.0,E3 0.0,E4 0.0,E5 0.0,E6 0.0}
DECL E6POS XSC_A2Return={X 232.779465,Y -108.546844,Z 1087.90991,A 154.999969,B 35.0000,C 179.999985,S 2,T 34,E1 0.0,E2 0.0,E3 0.0,E4 0.0,E5 0.0,E6 0.0}
DECL FDAT FSC_A2Return={TOOL_NO 0,BASE_NO 0,IPO_FRAME #BASE,POINT2[] " "}
DECL PDAT PPDAT15={VEL 100.000,ACC 60.0000,APO_DIST 500.000,APO_MODE #CDIS,GEAR_JERK 100.000,EXAX_IGN 0}
ENDDAT
